VAR_GLOBAL
	// XRTM1
	Serial_RXBuffer_XRTM1 : ComBuffer;
	Serial_TXBuffer_XRTM1 : ComBuffer;
END_VAR

(* stored: Version 1.1.0.1, ProductVersion 3.1.4022.18
   GVL GVL_COM_Buffers: Id {a8441f26-f9f8-4fbc-842d-41b6657e3ba7} *)
